(* Function that returns if an object is not initialized. *)
FUNCTION jog_manager_is_not_initialized : BOOL
VAR_IN_OUT
	CONVERSION_this:	jog_manager;	(* object reference *)
END_VAR

jog_manager_is_not_initialized:=NOT CONVERSION_this.CONVERSION_private.initialized;

END_FUNCTION

(* stored: Version 1.1.0.1, ProductVersion 3.1.4022.12
   POU jog_manager_is_not_initialized: Id {f9b86204-d3ac-460e-b38a-c550c69bb50e}, SpecialFunc None *)
